FUNCTION Convert_REAL_TO_ULINT : Hresult
VAR_INPUT
	in : REAL;
	out : REFERENCE TO ULINT;
END_VAR
VAR
	converted : ULINT;
END_VAR

converted := REAL_TO_ULINT(in);

IF (ULINT_TO_REAL(converted) <> in) THEN
	Convert_REAL_TO_ULINT := INCOMPATIBLE;
	RETURN;
END_IF

out := converted;

END_FUNCTION

(* stored: Version 1.1.0.1, ProductVersion 3.1.4024.12
   POU Convert_REAL_TO_ULINT: Id {0076797e-d393-45af-811f-9c8af0e61194}, SpecialFunc None *)
